Omron Sysmac Studio project Ethercat_Demo (Sysmac Studio 1.47.0.64008, StandardProject)

# Controller new_Controller_0: NX102-1220 version 1.38
Units and slaves: Node1 : ifm IO-Link Master AL1332(E001); 0 : IOL_4/4_I/O-Bytes(M1); 1 : Digital_IN(M9); 2 : Digital_OUT(M2); 3 : IOL_4/4_I/O-Bytes(M4); 4 : IOL_4/4_I/O-Bytes(M5); 5 : IOL_4/4_I/O-Bytes(M6); 6 : IOL_4/4_I/O-Bytes(M7); 7 : IOL_4/4_I/O-Bytes(M8); Node2 : AXL E EC DI8 DO8 M12 6P (E002)
Task PrimaryTask (priority 4, period or condition 2000): Program0

VAR_GLOBAL
    E002_RxPDO_Mapping_Digital_Outpu_Digital_Output_Bits_0_7_5000_01 : USINT;  (* at ECAT://node#2/RxPDO Mapping Digital Outpu_Digital Output Bits 0..7_5000_01 *)
    ifm_al1332_Slot2_DORxPDO_output_byte_0_7000_01 : USINT;  (* at ECAT://node#[1,2]/RxPDO_output byte 0_7000_01 *)
    ifm_al1332_Slot0_IolinkdataTxPDO_input_byte_0_6000_01 : USINT;  (* at ECAT://node#[1,0]/TxPDO_input byte 0_6000_01 *)
    ifm_al1332_Slot0_IolinkdataTxPDO_input_byte_1_6000_02 : USINT;  (* at ECAT://node#[1,0]/TxPDO_input byte 1_6000_02 *)
    E001_TxPDO_IO_Link_Port_Qualifie_IO_Link_Port_2_Qualifier_F101_02 : USINT;  (* at ECAT://node#1/TxPDO IO-Link Port Qualifie_IO-Link Port 2 Qualifier_F101_02 *)
    E001_TxPDO_IO_Link_Port_Qualifie_IO_Link_Port_1_Qualifier_F101_01 : USINT;  (* at ECAT://node#1/TxPDO IO-Link Port Qualifie_IO-Link Port 1 Qualifier_F101_01 *)
    E001_TxPDO_IO_Link_Port_Qualifie_IO_Link_Port_3_Qualifier_F101_03 : USINT;  (* at ECAT://node#1/TxPDO IO-Link Port Qualifie_IO-Link Port 3 Qualifier_F101_03 *)
    E001_TxPDO_IO_Link_Device_Status_IO_Link_Port_1_Status_F100_01 : USINT;  (* at ECAT://node#1/TxPDO IO-Link Device Status_IO-Link Port 1 Status_F100_01 *)
    E001_TxPDO_IO_Link_Device_Status_IO_Link_Port_2_Status_F100_02 : USINT;  (* at ECAT://node#1/TxPDO IO-Link Device Status_IO-Link Port 2 Status_F100_02 *)
    E001_TxPDO_IO_Link_Device_Status_IO_Link_Port_3_Status_F100_03 : USINT;  (* at ECAT://node#1/TxPDO IO-Link Device Status_IO-Link Port 3 Status_F100_03 *)
END_VAR

PROGRAM Program0
VAR
    MyTimer1 : TON;
    myStep : INT;
    Distance : INT;
    _temp : ULINT;
    ShiftWord1 : WORD;
    ShiftWord2 : WORD;
    AL1322_Qualifier : ARRAY[1..8] OF FB_IFM_AL1322_Qualifier;
    AL1322_Status : ARRAY[1..8] OF FB_IFM_AL1322_Status;
    myCounter : INT;
END_VAR
VAR_EXTERNAL
    E002_RxPDO_Mapping_Digital_Outpu_Digital_Output_Bits_0_7_5000_01 : USINT;
    ifm_al1332_Slot2_DORxPDO_output_byte_0_7000_01 : USINT;
    ifm_al1332_Slot0_IolinkdataTxPDO_input_byte_0_6000_01 : USINT;
    ifm_al1332_Slot0_IolinkdataTxPDO_input_byte_1_6000_02 : USINT;
    E001_TxPDO_IO_Link_Port_Qualifie_IO_Link_Port_1_Qualifier_F101_01 : USINT;
    E001_TxPDO_IO_Link_Port_Qualifie_IO_Link_Port_2_Qualifier_F101_02 : USINT;
    E001_TxPDO_IO_Link_Port_Qualifie_IO_Link_Port_3_Qualifier_F101_03 : USINT;
    E001_TxPDO_IO_Link_Device_Status_IO_Link_Port_1_Status_F100_01 : USINT;
    E001_TxPDO_IO_Link_Device_Status_IO_Link_Port_2_Status_F100_02 : USINT;
    E001_TxPDO_IO_Link_Device_Status_IO_Link_Port_3_Status_F100_03 : USINT;
END_VAR
//Qualifier
	AL1322_Qualifier[1](
		Qualifier:=E001_TxPDO_IO_Link_Port_Qualifie_IO_Link_Port_1_Qualifier_F101_01
		);
	AL1322_Qualifier[2](
		Qualifier:=E001_TxPDO_IO_Link_Port_Qualifie_IO_Link_Port_2_Qualifier_F101_02
		);
	AL1322_Qualifier[3](
		Qualifier:=E001_TxPDO_IO_Link_Port_Qualifie_IO_Link_Port_3_Qualifier_F101_03
		);
//Status
	AL1322_Status[1](
		Status:=E001_TxPDO_IO_Link_Device_Status_IO_Link_Port_1_Status_F100_01
		);
	AL1322_Status[2](
		Status:=E001_TxPDO_IO_Link_Device_Status_IO_Link_Port_2_Status_F100_02
		);	
	AL1322_Status[3](
		Status:=E001_TxPDO_IO_Link_Device_Status_IO_Link_Port_3_Status_F100_03
		);


IF myStep=0 AND AL1322_Qualifier[2].DI2 THEN

	MyTimer1(IN:=TRUE,pt:=T#1s);
	if MyTimer1.Q THEN
		myStep:=1;
		MyTimer1(IN:=False);
	END_IF;
END_IF;

if  AL1322_Qualifier[2].DI2 = false THEN
	myStep:=0;
END_IF;

CASE myStep OF
	
	
	0:
		E002_RxPDO_Mapping_Digital_Outpu_Digital_Output_Bits_0_7_5000_01:=16#00;
		ifm_al1332_Slot2_DORxPDO_output_byte_0_7000_01:=0;
	
	1:
		MyTimer1(In:=True, PT:=T#1s);
		E002_RxPDO_Mapping_Digital_Outpu_Digital_Output_Bits_0_7_5000_01:=16#FF;
		ifm_al1332_Slot2_DORxPDO_output_byte_0_7000_01:=1;
		IF MyTimer1.Q THEN
			myStep:=2;
			MyTimer1(In:=FALSE);
		END_IF;
	2:
		MyTimer1(In:=True, PT:=T#1s);
		E002_RxPDO_Mapping_Digital_Outpu_Digital_Output_Bits_0_7_5000_01:=16#00;
		ifm_al1332_Slot2_DORxPDO_output_byte_0_7000_01:=0;
		IF MyTimer1.Q THEN
			myStep:=1;
			MyTimer1(In:=FALSE);
		END_IF;
END_CASE;

Distance:=0;
if AL1322_Status[1].PortIsIOLink_OP THEN
	ShiftWord1:= SHL(
			 	USINT_TO_WORD(ifm_al1332_Slot0_IolinkdataTxPDO_input_byte_0_6000_01)
				,8
			);
	ShiftWord2:=USINT_TO_WORD(ifm_al1332_Slot0_IolinkdataTxPDO_input_byte_1_6000_02);


	Distance:=WORD_TO_INT(ShiftWord1 or ShiftWord2);

END_IF;
END_PROGRAM

FUNCTION_BLOCK FB_IFM_AL1322_Qualifier
VAR
    _Qualifier : WORD;
END_VAR
VAR_INPUT
    Qualifier : USINT;
END_VAR
VAR_OUTPUT
    DI4 : BOOL;
    DI2 : BOOL;
    PVO : BOOL;
    DACT : BOOL;
    DA : BOOL;
    PE : BOOL;
    PVI : BOOL;
END_VAR
_Qualifier:=USINT_TO_WORD(Qualifier);

DI4:=(_Qualifier & WORD#2#0000_0001)<>0;
DI2:=(_Qualifier & WORD#2#0000_0010)<>0;
PVO:=(_Qualifier & WORD#2#000_0100)<>0;

DACT:=(_Qualifier & WORD#2#0001_0000)<>0;
DA:=(_Qualifier & WORD#2#0010_0000)<>0;
PE:=(_Qualifier & WORD#2#0100_0000)<>0;
PVI:=(_Qualifier & WORD#2#1000_0000)<>0;
END_FUNCTION_BLOCK

FUNCTION_BLOCK FB_IFM_AL1322_Status
VAR
    _Status : WORD;
END_VAR
VAR_INPUT
    Status : USINT;
END_VAR
VAR_OUTPUT
    Error : BOOL;
    PortIsDeactivated : BOOL;
    PortIsDI : BOOL;
    PortIsDO : BOOL;
    PortIsIOLink_OP : BOOL;
    PortIsIOLink_STOP : BOOL;
    PortIsIOLink_PreOP : BOOL;
END_VAR
//Error
	_Status:=USINT_to_WORD(Status);
	Error:=(_Status & WORD#2#1111_0000)<>0;

//Port
	_Status:=_Status& WORD#2#0000_1111 ;
	PortIsDeactivated:=_Status = WORD#16#0;
	PortIsDI:=_Status=WORD#16#1;
	PortIsDO:=_Status = WORD#16#2;
	PortIsIOLink_OP:=_Status = WORD#16#3;
	PortIsIOLink_STOP:=_Status=WORD#16#4;
	PortIsIOLink_PreOP:=_Status=WORD#16#5;
	
END_FUNCTION_BLOCK